// TIA Portal V20 export
// export: Created 2025-12-01T14:57:21.1475372Z, ExportSetting None, DisplayName Totally Integrated Automation Portal, DisplayVersion V20 Update 3, DisplayName TIA Portal Openness, DisplayVersion V20 Update 3, DisplayName TIA Portal Version Control Interface, DisplayVersion V20 Update 3, DisplayName STEP 7 Professional, DisplayVersion V20 Update 3, DisplayName STEP 7 Safety, DisplayVersion V20 Update 2, DisplayName WinCC Basic/Comfort/Advanced, DisplayVersion V20 Update 3, DisplayName WinCC Professional, DisplayVersion V20 Update 3, DisplayName WinCC Unified, DisplayVersion V20 Update 3
DATA_BLOCK "DB2135_DB_AccesoMaq1"   // DB2135, F_DB
FAMILY : FPRI085e
VERSION : 0.0
// stored: AutoNumber false, InstanceOfName FB2142_F_AccesoMaquina, InstanceOfType FB
"FB2142_F_AccesoMaquina"
   // VAR_INPUT
   //    Maquina_OFF : Bool;
   //    PuertasAcceso_Cerradas : Bool;
   //    Acceso_Permitido : Bool;
   //    Peticion_Acceso : Bool;
   //    TIM_EsperaMaxima : Time;
   // END_VAR
   // VAR_OUTPUT
   //    Enclavamiento_Puertas : Bool;
   //    Puertas_OK : Bool;
   //    H_Acceso_Permitido : Bool;
   // END_VAR
   // VAR
   //    Temporizador_Espera { S7_SetPoint := 'True'} : TON;
   //    Puertas_ok_Aux : Bool;
   // END_VAR
BEGIN
END_DATA_BLOCK
